FUNCTION ATAN2 : LREAL
VAR_INPUT
	x: LREAL;
	y: LREAL;
END_VAR
VAR
END_VAR

IF x > 0 THEN
	ATAN2 := ATAN(y/x);
ELSIF x < 0 AND y > 0 THEN
	ATAN2 :=  ATAN(y/x) + pi;
ELSIF x < 0 AND y = 0 THEN
	ATAN2 := pi;
ELSIF x < 0 AND y < 0 THEN
	ATAN2 := ATAN(y/x) - pi;
ELSIF x = 0 AND y > 0 THEN
	ATAN2 := pi/2;
ELSIF x = 0 AND y < 0 THEN
    ATAN2 := -pi/2;
END_IF

END_FUNCTION

(* stored: Version 1.1.0.1, ProductVersion 3.1.4024.11
   POU ATAN2: Id {22eb7e13-a0a0-42b1-94a1-adee0d2bc3d4}, SpecialFunc None *)
